	            //Waiting for new postion from input, then setting end position
	            IF #sx_TrigPECInfeedD
	                AND #iqUDT_RATPositioning.Upper.StartPositionD <> 0
	                AND ((#sx_DataReceived
	                AND NOT #sx_DestinationC)
	                OR NOT #sx_DataReceived)
	            THEN
	                #sx_ServoInfeed := TRUE;
	                #iqUDT_RATPositioning.Upper.EndPosition := #iqUDT_RATPositioning.Upper.StartPositionD - #iUDT_Configuration.InfeedDDistance;
	                #sx_TrigPECInfeedD := FALSE;
	                #iqUDT_RATPositioning.Upper.StartPositionD := 0;
	                #iqUDT_RATPositioning.Upper.PositionRequired := FALSE;
	                #iqUDT_RATPositioning.Upper.Start := TRUE;
	                // If straight destination detected then use displacement mode
	            ELSIF #sx_TrigPECInfeedD
	                AND #sx_DataReceived
	                AND #sx_DestinationC
	            THEN
	                #si_UpperInfeedDistance := ABS(#iUDT_Configuration.InfeedDDistance / 10);
	                #sx_TrigPECInfeedD := FALSE;
	                #sx_DisplacementInfeed := TRUE;
	                #iqUDT_RATPositioning.Upper.StartPositionD := 0;
	                #iqUDT_RATPositioning.Upper.PositionRequired := FALSE;
	            END_IF;

	            //If position is reached, set ProductRecived
	            IF #sR_TRIG_UpperInfeedDone.Q
	                AND #sx_ServoInfeed
	            THEN
	                #sx_ProductReceivedUp := TRUE;
	                #iqUDT_RATPositioning.Upper.Start := FALSE;
	            END_IF;

	            // During upper infeeding count distance to end of RAT
	            IF #sx_UpperTransportIn AND
	                #sx_DisplacementInfeed
	                AND NOT #sx_ProductReceivedUp
	            THEN
	                #si_UpperInfeedDistance -= ABS(#iqUDT_UpperConveyorInterface.Displacement);
	                IF #si_UpperInfeedDistance <= 0
	                THEN
	                    #sx_ProductReceivedUp := TRUE;
	                END_IF;
	            END_IF;

	        END_REGION

	    END_REGION

	    REGION 7.4 - Infeed checked, go to infeed level
	        // Lower
	        IF #sx_AutomaticActive                                          // The device is automaticly started
	            AND #sx_Ready                                               // The device is ready to opereate
	            AND #sx_Active                                              // The sequence is started
	            AND #sx_InfeedCHK                                           // Step infeed check is active
	            AND ((#si_Conveyor = #ci_ConveyorA) OR #si_Conveyor = #ci_ConveyorB)// Infeed is on low level
	        THEN
	            #sx_MoveSectionDownInfeed := TRUE;                          // Move section down
	            #sx_InfeedCHK := FALSE;                                     // Reset step infeed check
	            #si_Step := 2;                                              // Set step number for diagnostic purposes
	            // Upper
	        ELSIF #sx_AutomaticActive                                       // The device is automaticly started
	            AND #sx_Ready                                               // The device is ready to opereate
	            AND #sx_Active                                              // The sequence is started
	            AND #sx_InfeedCHK                                           // Step infeed check is active
	            AND ((#si_Conveyor = #ci_ConveyorC) OR #si_Conveyor = #ci_ConveyorD) // Infeed is on high level
	        THEN
	            #sx_MoveSectionUpinfeed := TRUE;                            // Move section up
	            #sx_InfeedCHK := FALSE;                                     // Reset step infeed check
	            #si_Step := 2;                                              // Set step number for diagnostic purposes
	        END_IF;
	    END_REGION

	    REGION 7.5 - At infeed level, start infeed transport
	        // Lower
	        IF #sx_AutomaticActive                                          // The device is automaticly started
	            AND #sx_Ready                                               // The device is ready to opereate
	            AND #sx_Active                                              // The sequence is started
	            AND (#ix_SectionIsDown                                      // Section is actual down
	            OR (#sx_SectionDown                                         // or request to go down is set and configuration allows it
	            AND NOT #iUDT_Configuration.PositionVerification))
	            AND #sx_MoveSectionDownInfeed                               // Step move down to infeed was activated
	        THEN
	            #sx_MoveSectionDownInfeed := FALSE;                         // Reset step move down to infeed level
	            #sx_LowerTransportIn := TRUE;                               // Start infeed roller transport
	            #iqUDT_RATPositioning.Lower.PositionRequired := TRUE;
	            #sx_LowerRTR := TRUE;                                       // Set RTR to infeed until TIP gets active
	            #si_Step := 3;                                              // Set step number for diagnostic purposes
	            // Upper
	        ELSIF #sx_AutomaticActive                                       // The device is automaticly started
	            AND #sx_Ready                                               // The device is ready to opereate
	            AND #sx_Active                                              // The sequence is started
	            AND (#ix_SectionIsUp                                        // Section is actual up
	            OR (#sx_SectionUp                                           // or request to go up is set and configuration allows it
	            AND NOT #iUDT_Configuration.PositionVerification))
	            AND #sx_MoveSectionUpinfeed                                 // Step move up to infeed was activated
	            //     AND #iqUDT_UpperConveyorInterface.ActualSpeed = 0
	        THEN
	            #sx_MoveSectionUpinfeed := FALSE;                           // Reset step move up to infeed level
	            #sx_UpperTransportIn := TRUE;                               // Start infeed belt transport
	            #iqUDT_RATPositioning.Upper.PositionRequired := TRUE;
	            #sx_UpperRTR := TRUE;                                       // Set RTR to infeed until TIP gets active
	            #si_Step := 3;                                              // Set step number for diagnostic purposes

	        END_IF;
	    END_REGION

	    REGION 7.6 - Stop transport, wait for destnation

	        // Lower
	        IF #sx_AutomaticActive                                          // The device is automaticly started
	            AND #sx_Ready                                               // The device is ready to opereate
	            AND #sx_Active                                              // The sequence is started
	            AND #sx_LowerTransportIn                                    // Step infeed lower transport is active
	            AND (NOT #sx_PECFiltered OR NOT #iUDT_Configuration.ControlProductWithPEC)                                     // Position is occupied
	            AND #sx_ProductReceivedDown                                // Product available at the end of RAT

	        THEN
	            #sx_LowerTransportIn := FALSE;                              // Reset step infeed lower transport
	            #sx_LowerRTR := FALSE;                                      // Reset RTR signal for infeed conveyor
	            #sx_UpDown := TRUE;                                         // Wait for direction
	            #sx_ProductReceivedDown := FALSE;                           // Reset "product received" bit
	            #sx_ServoInfeed := FALSE;
	            #sx_DisplacementInfeed := FALSE;
	            #si_Step := 4;                                              // Set step number for diagnostic purposes

	            // Upper
	        ELSIF #sx_AutomaticActive                                       // The device is automaticly started
	            AND #sx_Ready                                               // The device is ready to opereate
	            AND #sx_Active                                              // The sequence is started
	            AND #sx_UpperTransportIn                                    // Step infeed belt transport is active
	            AND (NOT #sx_PECFiltered OR NOT #iUDT_Configuration.ControlProductWithPEC)                                      // Position is occupied
	            AND #sx_ProductReceivedUp                                  // Product available at the end of RAT
	        THEN
	            #sx_UpperTransportIn := FALSE;                              // Reset step infeed belttransport
	            #sx_UpperRTR := FALSE;                                      // Reset RTR signal for infeed conveyor
	            #sx_UpDown := TRUE;                                         // Wait for direction
	            #sx_ProductReceivedUp := FALSE;                             // Reset "product received" bit
	            #sx_ServoInfeed := FALSE;
	            #sx_DisplacementInfeed := FALSE;
	            #si_Step := 4;                                              // Set step number for diagnostic purposes

	        END_IF;
	    END_REGION

	    REGION 7.7 - Destination received, move to outfeed level
	        IF #sx_AutomaticActive                                                  // The device is automaticly started
	            AND #sx_Ready                                                       // The device is ready to opereate
	            AND #sx_Active                                                      // The sequence is started
	            AND #sx_UpDown                                                      // Wait for direction
	            AND #sx_DataReceived                                                // Direction is received
	        THEN
	            #sx_UpDown := FALSE;                                                // Wait for direction
	            #sx_MoveSectionDownOutfeed := #sx_DestinationA OR #sx_DestinationB; // Depending on outfeed conveyor section is moved to outfeed level
	            #sx_MoveSectionUpOutfeed := #sx_DestinationC OR #sx_DestinationD;   // Depending on outfeed conveyor section is moved to outfeed level
	            #si_Step := 5;                                                      // Set step number for diagnostic purposes
	        END_IF;
	    END_REGION


	    REGION 7.8 - At outfeed level, start outfeed transport
	        // Lower
	        IF #sx_AutomaticActive                                          // The device is automaticly started
	            AND #sx_Ready                                               // The device is ready to opereate
	            AND #sx_Active                                              // The sequence is started
	            AND #sx_MoveSectionDownOutfeed                              // Step move down to outfeed is active
	            AND (#ix_SectionIsDown                                      // Section is actual down
	            OR (#sx_SectionDown                                         // or request to go down is set and configuration allows it
	            AND NOT #iUDT_Configuration.PositionVerification))
	        THEN
	            #sx_MoveSectionDownOutfeed := FALSE;                        // Reset step move down to outfeed
	            #sx_LowerTransportOut := TRUE;                              // Start outfeed roller transport
	            #si_LowerOutfeedDistance := DINT_TO_INT(#iUDT_LowerConveyorConfiguration.Common.Length / 10);
	            #si_Step := 6;                                              // Set step number for diagnostic purposes
	            // Upper
	        ELSIF #sx_AutomaticActive                                       // The device is automaticly started
	            AND #sx_Ready                                               // The device is ready to opereate
	            AND #sx_Active                                              // The sequence is startede
	            AND #sx_MoveSectionUpOutfeed                                // Step move up to outfeed is active
	            AND (#ix_SectionIsUp                                        // Section is actual up
	            OR (#sx_SectionUp                                          // or request to go up is set and configuration allows it
	            AND NOT #iUDT_Configuration.PositionVerification))
	        THEN
	            #sx_MoveSectionUpOutfeed := FALSE;                          // Reset step move up to outfeed
	            #sx_UpperTransportOut := TRUE;                              // Start outfeed belt transport
	            #si_UpperOutfeedDistance := DINT_TO_INT(#iUDT_UpperConveyorConfiguration.Common.Length / 10);
	            #si_Step := 6;                                              // Set step number for diagnostic purposes
	        END_IF;
	    END_REGION


	    REGION 7.9 Outfeed product tracking

	        IF #sx_LowerTransportOut AND NOT #sx_ProductSentDown
	        THEN
	            #si_LowerOutfeedDistance -= ABS(#iqUDT_LowerConveyorInterface.Displacement);
	            IF #si_LowerOutfeedDistance <= 0
	            THEN
	                #sx_ProductSentDown := TRUE;
	            END_IF;
	        END_IF;

	        // Upper
	        IF #sx_UpperTransportOut AND NOT #sx_ProductSentUp
	        THEN
	            #si_UpperOutfeedDistance -= ABS(#iqUDT_UpperConveyorInterface.Displacement);
	            IF #si_UpperOutfeedDistance <= 0
	            THEN
	                #sx_ProductSentUp := TRUE;
	            END_IF;
	        END_IF;

	    END_REGION

	    REGION 7.9 - End sequence
	        IF #sx_AutomaticActive                                          // The device is automaticly started
	            AND #sx_Ready                                               // The device is ready to opereate
	            AND #sx_Active                                              // The sequence is started
	            AND ((#sx_LowerTransportOut AND #sx_ProductSentDown)        // Outfeed transport is active and Produce is away
	            OR (#sx_UpperTransportOut AND #sx_ProductSentUp))           // Outfeed transport is active and Produce is away
	            AND (#sx_PECFiltered OR NOT #iUDT_Configuration.ControlProductWithPEC)                                          // Position is cleared
	            OR #sFB_InfeedTimeout.qx_DelayedSignal                      // Operation time elapsed
	        THEN

	            // Reset all auxiliary bits and variables
	            #sx_LowerTransportOut := FALSE;
	            #sx_UpperTransportOut := FALSE;
	            #si_Conveyor := 0;
	            #sx_Active := FALSE;
	            #sx_DataReceived := FALSE;
	            #si_Step := 0;
	            IF #sx_DestinationA
	            THEN
	                #sx_DestinationA := FALSE;
	                #iqUDT_HandShakeConveyorA.GIN := 0;
	                #iqUDT_HandShakeConveyorA.NrOfPosToShift := 0;
	                #iqUDT_HandShakeConveyorA.TIP := FALSE;
	            END_IF;
	            IF #sx_DestinationB
	            THEN
	                #sx_DestinationB := FALSE;
	                #iqUDT_HandShakeConveyorB.GIN := 0;
	                #iqUDT_HandShakeConveyorB.NrOfPosToShift := 0;
	                #iqUDT_HandShakeConveyorB.TIP := FALSE;
	            END_IF;
	            IF #sx_DestinationC
	            THEN
	                #sx_DestinationC := FALSE;
	                #iqUDT_HandShakeConveyorC.GIN := 0;
	                #iqUDT_HandShakeConveyorC.NrOfPosToShift := 0;
	                #iqUDT_HandShakeConveyorC.TIP := FALSE;
	            END_IF;
	            IF #sx_DestinationD
	            THEN
	                #sx_DestinationD := FALSE;
	                #iqUDT_HandShakeConveyorD.GIN := 0;
	                #iqUDT_HandShakeConveyorD.NrOfPosToShift := 0;
	                #iqUDT_HandShakeConveyorD.TIP := FALSE;
	            END_IF;
	            #iqUDT_HandShakeConveyorA.RTR := FALSE;
	            #iqUDT_HandShakeConveyorB.RTR := FALSE;
	            #iqUDT_HandShakeConveyorC.RTR := FALSE;
	            #iqUDT_HandShakeConveyorD.RTR := FALSE;

	            #si_Destination := 0;
	            #sx_ProductReceivedDown := FALSE;
	            #sx_ProductReceivedUp := FALSE;
	            #sx_ProductSentDown := FALSE;
	            #sx_ProductSentUp := FALSE;
	            #iqUDT_RATPositioning.Lower.ResetPosition := TRUE;
	            #iqUDT_RATPositioning.Upper.ResetPosition := TRUE;
	            #iqUDT_RATPositioning.Lower.StartPositionA := 0;
	            #iqUDT_RATPositioning.Lower.StartPositionB := 0;
	            #iqUDT_RATPositioning.Upper.StartPositionC := 0;
	            #iqUDT_RATPositioning.Upper.StartPositionD := 0;
	            #iqUDT_RATPositioning.Lower.PositionRequired := FALSE;
	            #iqUDT_RATPositioning.Upper.PositionRequired := FALSE;

	            // Move to configured default position
	            IF #iUDT_Configuration.DefaultPosition = #ci_DefaultPositionUp
	                AND #ix_SectionIsUp                                     // Section is actual up
	                AND #sa_FiFo[1] = 0
	            THEN
	                #sx_MoveSectiondownEnd := TRUE;                         // Then move down to infeed
	            END_IF;
	            IF #iUDT_Configuration.DefaultPosition = #ci_DefaultPositiondown
	                AND #ix_SectionIsDown                                   // Section is actual down
	                AND #sa_FiFo[1] = 0
	            THEN
	                #sx_MoveSectionUpEnd := TRUE;                           // Then move down to infeed
	            END_IF;
	        END_IF;
	        // Reset when on position
	        IF #sx_MoveSectionUpEnd                                         // Reset Up request when up
	            AND #ix_SectionIsUp
	        THEN
	            #sx_MoveSectionUpEnd := False;
	        END_IF;

	        IF #sx_MoveSectiondownEnd                                       // Reset down request when down
	            AND #ix_SectionIsDown
	        THEN
	            #sx_MoveSectiondownEnd := False;
	        END_IF;

	    END_REGION
	END_REGION

	REGION 8 - Output
	    REGION 8.1 - Lifting device

	        // Conditions to move sention down
	        #sx_SectionDown := (#sx_AutomaticActive
	        AND
	        ((#sx_MoveSectionDownInfeed OR #sx_MoveSectionDownOutfeed OR #sx_MoveSectiondownEnd))
	        OR (#sx_ManualModeActive AND #sx_ManualGoDown));
	        // Conditions to move sention up
	        #sx_SectionUp := (#sx_AutomaticActive
	        AND
	        ((#sx_MoveSectionUpinfeed OR #sx_MoveSectionUpOutfeed OR #sx_MoveSectionUpEnd))
	        OR (#sx_ManualModeActive AND #sx_ManualGoUp));

	        // Write valve outputs
	        IF #sx_SectionUp
	        THEN
	            #qx_PopupControl := TRUE;
	        ELSIF #sx_SectionDown
	        THEN
	            #qx_PopupControl := FALSE;
	        END_IF;

	    END_REGION

	    REGION 8.2 - Lower conveyor

	        // Run forward
	        #tx_LowerConveyorRunFwd :=
	        ((#sx_LowerTransportIn AND (#si_Conveyor = #ci_ConveyorA) AND #ix_ConveyorAAuto)                                    // Transport in and transporting from infeed A
	        OR (#sx_LowerTransportOut AND #sx_DestinationB AND #iqUDT_HandShakeConveyorB.RTR))                      // Transport out and RTR is received
	        AND #sx_AutomaticActive;

	        // Run reverse
	        #tx_LowerConveyorRunRvs :=
	        ((#sx_LowerTransportIn AND (#si_Conveyor = #ci_ConveyorB) AND #ix_ConveyorBAuto)                                     // Transport in and transporting from infeed B
	        OR (#sx_LowerTransportOut AND #sx_DestinationA AND #iqUDT_HandShakeConveyorA.RTR))                      // Transport out AND RTR is received
	        AND #sx_AutomaticActive;
	        // Handshake RTR mapping
	        #sUDT_HandshakeUpLowerConveyor.RTR := #tx_LowerConveyorRunRvs;
	        #sUDT_HandshakeLowerConveyor.RTR := #tx_LowerConveyorRunFwd;

	        IF #tx_LowerConveyorRunRvs THEN
	            #sx_ReverseLower := TRUE;
	        END_IF;

	        IF #tx_LowerConveyorRunFwd THEN
	            #sx_ReverseLower := FALSE;
	        END_IF;

	        // Control lower conveyor with FB_Conveyor block
	        #sFB_Conveyor_LowerConveyor(iUDT_ConveyorConfiguration := #iUDT_LowerConveyorConfiguration,
	                                    ix_SafetyOk := #ix_SafetyOk,
	                                    ix_24vOk := #ix_24vOk,
	                                    ix_400vOk := #ix_400vOk,
	                                    ix_HardwareOk := #ix_HardwareOk,
	                                    ix_ReverseDirection := #sx_ReverseLower,
	                                    ix_ResetEnergySave := TRUE,
	                                    qUDT_HMIStatus => #qUDT_HMIConveyorStatus,
	                                    qUDT_Status => #qUDT_ConveyorStatus,
	                                    iqUDT_EquipmentControl := #iqUDT_EquipmentControl,
	                                    iqUDT_ConveyorCommand := #iqUDT_ConveyorCommand,
	                                    iqUDT_ConveyorInterface := #iqUDT_LowerConveyorInterface,
	                                    iqUDT_HandShakeUp := #sUDT_HandshakeUpLowerConveyor,
	                                    iqUDT_HandShake := #sUDT_HandshakeLowerConveyor,
	                                    iqUDT_Statistics := #iqUDT_ConveyorStatistics);

	    END_REGION

	    REGION 8.3 - Upper conveyor

	        // Run forward
	        #tx_UpperConveyorRunFwd :=
	        ((#sx_UpperTransportIn AND (#si_Conveyor = #ci_ConveyorC) AND #ix_ConveyorCAuto)                                                  // Transport in and transporting from infeed C c
	        OR (#sx_UpperTransportOut AND #sx_DestinationD AND #iqUDT_HandShakeConveyorD.RTR))             // Transport out and RTR is received
	        AND #sx_AutomaticActive;

	        // Run reverse
	        #tx_UpperConveyorRunRvs :=
	        ((#sx_UpperTransportIn AND (#si_Conveyor = #ci_ConveyorD) AND #ix_ConveyorDAuto)                                                   // Transport in and transporting from infeed D
	        OR (#sx_UpperTransportOut AND #sx_DestinationC AND #iqUDT_HandShakeConveyorC.RTR))              // Transport out and RTR is received
	        AND #sx_AutomaticActive;

	        // Handshake RTR mapping
	        #sUDT_HandshakeUpUpperConveyor.RTR := #tx_UpperConveyorRunRvs;
	        #sUDT_HandshakeUpperConveyor.RTR := #tx_UpperConveyorRunFwd;


	        // MAnual mode mapping from RAT structure
	        #tUDT_ConveyorCommandUpper.ManualMode := #iqUDT_RATCommand.ManualMode;
	        #tUDT_ConveyorCommandUpper.ManualStartStop := #iqUDT_RATCommand.ManualStartStop;
	        #tUDT_ConveyorCommandUpper.ManualFullSpeed := #iqUDT_RATCommand.ManualFullSpeed;
	        #tUDT_ConveyorCommandUpper.ManualSpeed := #iqUDT_RATCommand.ManualSpeed;
	        #tUDT_ConveyorCommandUpper.ManualJog := #iqUDT_RATCommand.ManualJog;
	        #tUDT_ConveyorCommandUpper.Reverse := #iqUDT_RATCommand.Reverse;

	        IF #tx_UpperConveyorRunRvs
	        THEN
	            #sx_ReverseUpper := TRUE;
	        END_IF;

	        IF #tx_UpperConveyorRunFwd
	        THEN
	            #sx_ReverseUpper := FALSE;
	        END_IF;

	        // Control pop-up conveyor with FB_Conveyor block
	        #sFB_Conveyor_UpperConveyor(iUDT_ConveyorConfiguration := #iUDT_UpperConveyorConfiguration,
	                                    ix_SafetyOk := #ix_SafetyOk,
	                                    ix_24vOk := #ix_24vOk,
	                                    ix_400vOk := #ix_400vOk,
	                                    ix_HardwareOk := #ix_HardwareOk,
	                                    ix_ReverseDirection := #sx_ReverseUpper,
	                                    ix_ExternalRequestDieBack := FALSE,
	                                    ix_ResetEnergySave := TRUE,
	                                    qUDT_HMIStatus => #tUDT_HMIStatus,
	                                    qUDT_Status => #tUDT_CommonStatus,
	                                    iqUDT_EquipmentControl := #iqUDT_EquipmentControl,
	                                    iqUDT_ConveyorCommand := #tUDT_ConveyorCommandUpper,
	                                    iqUDT_ConveyorInterface := #iqUDT_UpperConveyorInterface,
	                                    iqUDT_HandShakeUp := #sUDT_HandshakeUpUpperConveyor,
	                                    iqUDT_HandShake := #sUDT_HandshakeUpperConveyor,
	                                    iqUDT_Statistics := #tUDT_ConveyorStatistics);

	        // Manual mode mapping from conveyor to RAT
	        #iqUDT_RATCommand.ManualMode := #tUDT_ConveyorCommandUpper.ManualMode;
	        #iqUDT_RATCommand.ManualStartStop := #tUDT_ConveyorCommandUpper.ManualStartStop;
	        #iqUDT_RATCommand.ManualFullSpeed := #tUDT_ConveyorCommandUpper.ManualFullSpeed;
	        #iqUDT_RATCommand.ManualSpeed := #tUDT_ConveyorCommandUpper.ManualSpeed;
	        #iqUDT_RATCommand.ManualJog := #tUDT_ConveyorCommandUpper.ManualJog;

	    END_REGION


	    REGION 8.4 - Handshake in-outfeed conveyors

	        #iqUDT_HandShakeConveyorA.RTR := FALSE;
	        #iqUDT_HandShakeConveyorB.RTR := FALSE;
	        #iqUDT_HandShakeConveyorC.RTR := FALSE;
	        #iqUDT_HandShakeConveyorD.RTR := FALSE;

	        IF (#si_Conveyor = 1)
	        THEN
	            // Infeed conveyor low level
	            #iqUDT_HandShakeConveyorA.CascadeStartUp := #sx_AutomaticActive;
	            #iqUDT_HandShakeConveyorA.RTR := (#sx_LowerRTR OR #iqUDT_HandShakeConveyorA.TIP) AND #sx_AutomaticActive;
	            #iqUDT_HandShakeConveyorA.ResetEnergySave := false;

	            IF #sx_LowerTransportIn
	            THEN
	                IF #iqUDT_HandShakeConveyorA.GIN <> 0
	                THEN                          // Save gin number in buffer
	                    #sUDT_HandshakeBuffer.GIN := #iqUDT_HandShakeConveyorA.GIN;
	                END_IF;

	                // Count number position to shift in buffer
	                #sUDT_HandshakeBuffer.NrOfPosToShift += #iqUDT_HandShakeConveyorA.NrOfPosToShift;
	                #iqUDT_HandShakeConveyorA.NrOfPosToShift := 0;
	            END_IF;

	        ELSE
	            // Outfeed conveyor low level
	            #qx_ExternalSendRequestA := #sx_DestinationA AND NOT #sFB_PEC.qx_PECFiltered;// AND #sx_LowerTransportOut;
	            IF #sx_LowerTransportOut AND #sx_DestinationA
	            THEN
	                IF #sR_TRIG_LowerOutfeedRunning.Q
	                THEN
	                    #iqUDT_HandShakeConveyorA.GIN := #sUDT_HandshakeBuffer.GIN;
	                    #iqUDT_HandShakeConveyorA.NrOfPosToShift := #sUDT_HandshakeBuffer.NrOfPosToShift;
	                    #sUDT_HandshakeBuffer.GIN := 0;
	                    #sUDT_HandshakeBuffer.NrOfPosToShift := 0;
	                END_IF;

	                IF #ix_PEC
	                THEN
	                    #iqUDT_HandShakeConveyorA.GIN := 0;
	                    #iqUDT_HandShakeConveyorA.NrOfPosToShift := 0;
	                END_IF;
	            END_IF;

	        END_IF;

	        IF (#si_Conveyor = 2)
	        THEN
	            // Infeed conveyor low level
	            #iqUDT_HandShakeConveyorB.CascadeStartUp := #sx_AutomaticActive;
	            #iqUDT_HandShakeConveyorB.RTR := (#sx_LowerRTR OR #iqUDT_HandShakeConveyorB.TIP) AND #sx_AutomaticActive;
	            #iqUDT_HandShakeConveyorB.ResetEnergySave := false;
	            IF #sx_LowerTransportIn
	            THEN
	                IF #iqUDT_HandShakeConveyorB.GIN <> 0
	                THEN
	                    #sUDT_HandshakeBuffer.GIN := #iqUDT_HandShakeConveyorB.GIN;
	                END_IF;

	                #sUDT_HandshakeBuffer.NrOfPosToShift += #iqUDT_HandShakeConveyorB.NrOfPosToShift;
	                #iqUDT_HandShakeConveyorB.NrOfPosToShift := 0;
	            END_IF;
	        ELSE
	            // Outfeed conveyor low level
	            #qx_ExternalSendRequestB := #sx_DestinationB AND NOT #sFB_PEC.qx_PECFiltered;// AND #sx_LowerTransportOut;
	            IF #sx_DestinationB AND #sx_LowerTransportOut
	            THEN
	                IF #sR_TRIG_LowerOutfeedRunning.Q
	                THEN
	                    #iqUDT_HandShakeConveyorB.GIN := #sUDT_HandshakeBuffer.GIN;
	                    #iqUDT_HandShakeConveyorB.NrOfPosToShift := #sUDT_HandshakeBuffer.NrOfPosToShift;
	                    #sUDT_HandshakeBuffer.GIN := 0;
	                    #sUDT_HandshakeBuffer.NrOfPosToShift := 0;
	                END_IF;

	                IF #ix_PEC
	                THEN
	                    #iqUDT_HandShakeConveyorB.GIN := 0;
	                    #iqUDT_HandShakeConveyorB.NrOfPosToShift := 0;

	                END_IF;

	            END_IF;
	        END_IF;

	        IF (#si_Conveyor = 3)
	        THEN
	            // Infeed conveyor high level
	            #iqUDT_HandShakeConveyorC.CascadeStartUp := #sx_AutomaticActive;
	            #iqUDT_HandShakeConveyorC.RTR := (#sx_UpperRTR OR #iqUDT_HandShakeConveyorC.TIP) AND #sx_AutomaticActive;
	            #iqUDT_HandShakeConveyorC.ResetEnergySave := false;
	            IF #sx_UpperTransportIn
	            THEN
	                IF #iqUDT_HandShakeConveyorC.GIN <> 0
	                THEN
	                    #sUDT_HandshakeBuffer.GIN := #iqUDT_HandShakeConveyorC.GIN;
	                END_IF;

	                #sUDT_HandshakeBuffer.NrOfPosToShift += #iqUDT_HandShakeConveyorC.NrOfPosToShift;
	                #iqUDT_HandShakeConveyorC.NrOfPosToShift := 0;
	            END_IF;
	        ELSE
	            // Outfeed conveyor high level
	            #qx_ExternalSendRequestC := #sx_DestinationC AND NOT #sFB_PEC.qx_PECFiltered;// AND #sx_LowerTransportOut;
	            IF #sx_DestinationC AND #sx_UpperTransportOut
	            THEN
	                IF #sR_TRIG_UpperOutfeedRunning.Q
	                THEN
	                    #iqUDT_HandShakeConveyorC.GIN := #sUDT_HandshakeBuffer.GIN;
	                    #iqUDT_HandShakeConveyorC.NrOfPosToShift := #sUDT_HandshakeBuffer.NrOfPosToShift;
	                    #sUDT_HandshakeBuffer.GIN := 0;
	                    #sUDT_HandshakeBuffer.NrOfPosToShift := 0;
	                END_IF;
	                IF #ix_PEC
	                THEN
	                    #iqUDT_HandShakeConveyorC.GIN := 0;
	                    #iqUDT_HandShakeConveyorC.NrOfPosToShift := 0;
	                END_IF;

	            END_IF;

	        END_IF;

	        IF (#si_Conveyor = 4)
	        THEN
	            // Infeed conveyor high level
	            #iqUDT_HandShakeConveyorD.CascadeStartUp := #sx_AutomaticActive;
	            #iqUDT_HandShakeConveyorD.RTR := (#sx_UpperRTR OR #iqUDT_HandShakeConveyorD.TIP) AND #sx_AutomaticActive;
	            #iqUDT_HandShakeConveyorD.ResetEnergySave := false;
	            IF #sx_UpperTransportIn
	            THEN
	                IF #iqUDT_HandShakeConveyorD.GIN <> 0
	                THEN
	                    #sUDT_HandshakeBuffer.GIN := #iqUDT_HandShakeConveyorD.GIN;
	                END_IF;

	                #sUDT_HandshakeBuffer.NrOfPosToShift += #iqUDT_HandShakeConveyorD.NrOfPosToShift;
	                #iqUDT_HandShakeConveyorD.NrOfPosToShift := 0;
	            END_IF;
	        ELSE
	            // Outfeed conveyor high level
	            #qx_ExternalSendRequestD := #sx_DestinationD AND NOT #sFB_PEC.qx_PECFiltered;// AND #sx_LowerTransportOut;
	            IF #sx_DestinationD AND #sx_UpperTransportOut
	            THEN
	                IF #sR_TRIG_UpperOutfeedRunning.Q
	                THEN
	                    #iqUDT_HandShakeConveyorD.GIN := #sUDT_HandshakeBuffer.GIN;
	                    #iqUDT_HandShakeConveyorD.NrOfPosToShift := #sUDT_HandshakeBuffer.NrOfPosToShift;
	                    #sUDT_HandshakeBuffer.GIN := 0;
	                    #sUDT_HandshakeBuffer.NrOfPosToShift := 0;
	                END_IF;

	                IF #ix_PEC
	                THEN
	                    #iqUDT_HandShakeConveyorD.GIN := 0;
	                    #iqUDT_HandShakeConveyorD.NrOfPosToShift := 0;
	                END_IF;

	            END_IF;

	        END_IF;

	    END_REGION

	    REGION 8.5 - Blade stop EoS
	        // If blade stop is available then handle valve
	        IF #iUDT_Configuration.BladeStopEoS
	        THEN
	            // Use blade stop if product is comming from A to side destination
	            IF #si_Conveyor = #ci_ConveyorA AND (#sx_DestinationC OR #sx_DestinationD) AND #sx_LowerTransportIn
	            THEN
	                #sx_BladeStopEoSControl := TRUE;
	            END_IF;
	            IF NOT #sx_LowerTransportIn
	            THEN
	                #sx_BladeStopEoSControl := FALSE;
	            END_IF;
	            #iqUDT_BladeStopEoSInterface.Open := #sx_BladeStopEoSControl;
	        END_IF;

	    END_REGION

	    REGION 8.6 - Blade stop BoS
	        IF #iUDT_Configuration.BladeStopBoS
	        THEN
	            // Use blade stop if product is comming from B to side destination
	            IF #si_Conveyor = #ci_ConveyorB AND (#sx_DestinationC OR #sx_DestinationD) AND #sx_LowerTransportIn
	            THEN
	                #sx_BladeStopBoSControl := TRUE;
	            END_IF;
	            IF NOT #sx_LowerTransportIn
	            THEN
	                #sx_BladeStopBoSControl := FALSE;
	            END_IF;
	            #iqUDT_BladeStopBoSInterface.Open := #sx_BladeStopBoSControl;
	        END_IF;

	    END_REGION

	END_REGION

	REGION 9 - PEC
	    // Use displacement from both interfaces - lower and upper
	    #tUDT_ConveyorInterface := #iqUDT_UpperConveyorInterface;
	    #tUDT_ConveyorInterface.Displacement := #iqUDT_UpperConveyorInterface.Displacement + #iqUDT_LowerConveyorInterface.Displacement;

	    // PEC handling
	    #sFB_PEC(ix_PEC := #ix_PEC,
	             iUDT_PECConfiguration := #iUDT_PECConfiguration,
	             qUDT_HMIStatus => #qUDT_HMIPECStatus,
	             iqUDT_ConveyorInterface := #tUDT_ConveyorInterface,
	             iqUDT_PECStatistics := #iqUDT_PECStatistics);

	    // copy error to both intefaces - lower and upper
	    #iqUDT_UpperConveyorInterface.InternalErrorPEC := #iqUDT_UpperConveyorInterface.InternalErrorPEC OR #tUDT_ConveyorInterface.InternalErrorPEC;
	    #iqUDT_LowerConveyorInterface.InternalErrorPEC := #iqUDT_LowerConveyorInterface.InternalErrorPEC OR #tUDT_ConveyorInterface.InternalErrorPEC;

	END_REGION

	REGION 9 - Status

	    // Status update
	    #sUDT_HMIStatus.Specific.Down := #ix_SectionIsDown AND NOT #ix_SectionIsUp;
	    #sUDT_HMIStatus.Specific.Up := #ix_SectionIsUp AND NOT #ix_SectionIsDown;
	    #sUDT_HMIStatus.Specific.Reverse := #tUDT_HMIStatus.Specific.Reverse;
	    #sUDT_HMIStatus.Status := #tUDT_HMIStatus.Status;

	    #sUDT_CommonStatus.SafetyStop := NOT #ix_SafetyOk AND #ix_HardwareOk;
	    #sUDT_CommonStatus.Stopped := NOT #sx_Ready OR NOT #sx_AutomaticActive OR #tUDT_CommonStatus.Stopped;
	    #sUDT_CommonStatus.AutoON := #sx_Ready AND #sx_AutomaticActive AND #tUDT_CommonStatus.AutoON;
	    #sUDT_CommonStatus.Manual := #sx_ManualModeActive;
	    #sUDT_CommonStatus.ManualRun := #sx_ManualModeActive AND #sUDT_CommonStatus.Running;
	    #sUDT_CommonStatus.Running := #tUDT_CommonStatus.Running;

	    #qUDT_RATStatus := #sUDT_CommonStatus;
	    #qUDT_HMIRATStatus := #sUDT_HMIStatus;

	END_REGION

	REGION 10 - Statistics

	    REGION 10.1 - Air pressure fault
	        // Update statistics if error is active or statistics reset detected
	        IF #sUDT_HMIStatus.Specific.ErrAirpressureNotOk OR #iqUDT_EquipmentControl.Command.ResetData      // Reset statistics
	        THEN

	            "FC_Statistics"(ix_Reset := #iqUDT_EquipmentControl.Command.ResetData,  // Reset statistics input
	                            ix_Activate := #sUDT_HMIStatus.Specific.ErrAirpressureNotOk,
	                            ix_RTrigActivate := #sR_TRIG_AirPressureFault.Q,            // Statistics active trigger
	                            iqUDT_Statistics := #iqUDT_RATStatistics.AirPressure);

	        END_IF;

	    END_REGION

	    REGION 10.2 - Device up time

	        // Conveyor up is when conveyor is not in manual mode and has an error
	        IF #sx_DivertUpRunTimeErr OR #iqUDT_EquipmentControl.Command.ResetData      // Reset statistics
	        THEN

	            "FC_Statistics"(ix_Reset := #iqUDT_EquipmentControl.Command.ResetData,  // Reset statistics input
	                            ix_Activate := #sx_DivertUpRunTimeErr, // Activate statistics functions input
	                            ix_RTrigActivate := #sR_TRIG_DivertUpError.Q,          // Statistics active trigger
	                            iqUDT_Statistics := #iqUDT_RATStatistics.DivertUpError);   // Statistics values output

	        END_IF;

	    END_REGION

	    REGION 10.3 - Device down time

	        // Conveyor down is when conveyor is not in manual mode and has an error
	        IF #sx_DivertDownRunTimeErr OR #iqUDT_EquipmentControl.Command.ResetData      // Reset statistics
	        THEN

	            "FC_Statistics"(ix_Reset := #iqUDT_EquipmentControl.Command.ResetData,  // Reset statistics input
	                            ix_Activate := #sx_DivertDownRunTimeErr, // Activate statistics functions input
	                            ix_RTrigActivate := #sR_TRIG_DivertDownError.Q,          // Statistics active trigger
	                            iqUDT_Statistics := #iqUDT_RATStatistics.DivertDownError);   // Statistics values output

	        END_IF;

	    END_REGION

	    REGION 10.4 - Conveyor statistics
	        // Copy statistics from conveyor block
	        #iqUDT_RATStatistics.ConveyorDown := #tUDT_ConveyorStatistics.ConveyorDown;
	        #iqUDT_RATStatistics.ConveyorStop := #tUDT_ConveyorStatistics.ConveyorStop;
	        #iqUDT_RATStatistics.ConveyorUp := #tUDT_ConveyorStatistics.ConveyorUp;

	    END_REGION

	END_REGION

	REGION 11 - Report to control block
	    // Function to manage report between control block and conveyor block
	    "FC_EquipmentReport"(iUDT_Status := #sUDT_CommonStatus,
	                         iqUDT_Control := #iqUDT_EquipmentControl);

	END_REGION

	REGION 12 - Internal errors and warnings reset

	    REGION 12.1 Infeed timeout
	        // Infeed stuck, timeout calculation
	        #sFB_InfeedTimeout(iudi_OnDelayTime := #iUDT_Configuration.InfeedTimeout,
	                           ix_SignalToDelay := #si_Step = 3 AND (#sx_ProductReceivedDown OR #sx_ProductReceivedUp));

	    END_REGION

	    REGION 12.2 Reactivation
	        // Reactivate conveyor 1 if request is active and no register find
	        #sFB_ConveyorAReactivation(iudi_OnDelayTime := #iUDT_Configuration.ReactivationTime,
	                                   ix_SignalToDelay := #ix_ExternalReceiveRequestA AND #ix_ConveyorAAuto);

	        IF #sFB_ConveyorAReactivation.qx_DelayedSignal AND NOT (#si_Conveyor = 1)
	        THEN
	            #sx_ReactivateA := TRUE;
	            FOR #si_LoopArrayCount := 1 TO #ci_FiFoLength DO

	                IF #sa_FiFo[#si_LoopArrayCount] = 1
	                THEN
	                    #sx_ReactivateA := FALSE;
	                END_IF;

	            END_FOR;

	        END_IF;
	        // Reactivate conveyor 1 if request is active and no register find
	        #sFB_ConveyorBReactivation(iudi_OnDelayTime := #iUDT_Configuration.ReactivationTime,
	                                   ix_SignalToDelay := #ix_ExternalReceiveRequestB AND #ix_ConveyorBAuto);

	        IF #sFB_ConveyorBReactivation.qx_DelayedSignal AND NOT (#si_Conveyor = 2)
	        THEN
	            #sx_ReactivateB := TRUE;
	            FOR #si_LoopArrayCount := 1 TO #ci_FiFoLength DO

	                IF #sa_FiFo[#si_LoopArrayCount] = 2
	                THEN
	                    #sx_ReactivateB := FALSE;
	                END_IF;

	            END_FOR;

	        END_IF;
	        // Reactivate conveyor 1 if request is active and no register find
	        #sFB_ConveyorCReactivation(iudi_OnDelayTime := #iUDT_Configuration.ReactivationTime,
	                                   ix_SignalToDelay := #ix_ExternalReceiveRequestC AND #ix_ConveyorCAuto);

	        IF #sFB_ConveyorCReactivation.qx_DelayedSignal AND NOT (#si_Conveyor = 3)
	        THEN
	            #sx_ReactivateC := TRUE;
	            FOR #si_LoopArrayCount := 1 TO #ci_FiFoLength DO

	                IF #sa_FiFo[#si_LoopArrayCount] = 3
	                THEN
	                    #sx_ReactivateC := FALSE;
	                END_IF;

	            END_FOR;

	        END_IF;
	        // Reactivate conveyor 1 if request is active and no register find
	        #sFB_ConveyorDReactivation(iudi_OnDelayTime := #iUDT_Configuration.ReactivationTime,
	                                   ix_SignalToDelay := #ix_ExternalReceiveRequestD AND #ix_ConveyorDAuto);

	        IF #sFB_ConveyorDReactivation.qx_DelayedSignal AND NOT (#si_Conveyor = 4)
	        THEN
	            #sx_ReactivateD := TRUE;
	            FOR #si_LoopArrayCount := 1 TO #ci_FiFoLength DO

	                IF #sa_FiFo[#si_LoopArrayCount] = 4
	                THEN
	                    #sx_ReactivateD := FALSE;
	                END_IF;

	            END_FOR;

	        END_IF;

	    END_REGION

	END_REGION
END_FUNCTION_BLOCK

DATA_BLOCK "DB_FIFOLostGIN"
TITLE = DB_FIFO
{ S7_Optimized_Access := 'TRUE' }
AUTHOR : MHSE
FAMILY : GeneralSystemFunctions
VERSION : 3.0
NON_RETAIN
//Data block to store FIFO registers.
   VAR RETAIN
      Header { ExternalAccessible := 'False'; ExternalVisible := 'False'; ExternalWritable := 'False'; S7_SetPoint := 'False'} : "UDT_FifoHeader";   // FIFO Header
      Data { ExternalAccessible := 'False'; ExternalVisible := 'False'; ExternalWritable := 'False'} : Array[0..199] of Int;   // FIFO data buffer
   END_VAR
   VAR
      Header_1 { ExternalAccessible := 'False'; ExternalVisible := 'False'; ExternalWritable := 'False'; S7_SetPoint := 'False'} : "UDT_FifoHeader";
      Data_1 { ExternalAccessible := 'False'; ExternalVisible := 'False'; ExternalWritable := 'False'} : Array[0..199] of Int;
      Header_2 { ExternalAccessible := 'False'; ExternalVisible := 'False'; ExternalWritable := 'False'; S7_SetPoint := 'False'} : "UDT_FifoHeader";
      Data_2 { ExternalAccessible := 'False'; ExternalVisible := 'False'; ExternalWritable := 'False'} : Array[0..199] of Int;
      Header_3 { ExternalAccessible := 'False'; ExternalVisible := 'False'; ExternalWritable := 'False'; S7_SetPoint := 'False'} : "UDT_FifoHeader";
      Data_3 { ExternalAccessible := 'False'; ExternalVisible := 'False'; ExternalWritable := 'False'} : Array[0..199] of Int;
      Header_4 { ExternalAccessible := 'False'; ExternalVisible := 'False'; ExternalWritable := 'False'; S7_SetPoint := 'False'} : "UDT_FifoHeader";
      Data_4 { ExternalAccessible := 'False'; ExternalVisible := 'False'; ExternalWritable := 'False'} : Array[0..199] of Int;
      Header_5 { ExternalAccessible := 'False'; ExternalVisible := 'False'; ExternalWritable := 'False'; S7_SetPoint := 'False'} : "UDT_FifoHeader";
      Data_5 { ExternalAccessible := 'False'; ExternalVisible := 'False'; ExternalWritable := 'False'} : Array[0..199] of Int;
      Header_6 { ExternalAccessible := 'False'; ExternalVisible := 'False'; ExternalWritable := 'False'; S7_SetPoint := 'False'} : "UDT_FifoHeader";
      Data_6 { ExternalAccessible := 'False'; ExternalVisible := 'False'; ExternalWritable := 'False'} : Array[0..199] of Int;
   END_VAR


BEGIN

END_DATA_BLOCK

FUNCTION_BLOCK "FB_CognexDM260"
{ S7_Optimized_Access := 'TRUE' }
VERSION : 0.1
// ATTRIBUTES
// AUTO_NUMBER = True
// BLOCK_NUMBER = 263
// END_ATTRIBUTES
   VAR_INPUT
      iUDT_CognexDM260_IN { ExternalAccessible := 'False'; ExternalVisible := 'False'; ExternalWritable := 'False'} : "UDT_CognexDM260_IN";   // Data from camera
      ix_Trigger { ExternalAccessible := 'False'; ExternalVisible := 'False'; ExternalWritable := 'False'} : Bool;   // Trigger - Activate barcode scanning inside this function
   END_VAR

   VAR_OUTPUT
      qUDT_CognexDM260_OUT { ExternalAccessible := 'False'; ExternalVisible := 'False'; ExternalWritable := 'False'} : "UDT_CognexDM260_OUT";   // Data send to camera
      qs_Barcode { ExternalAccessible := 'False'; ExternalVisible := 'False'; ExternalWritable := 'False'} : String;
      qw_RetVal { ExternalAccessible := 'False'; ExternalVisible := 'False'; ExternalWritable := 'False'} : Word;   // Error code (W#16#...): A - TimeOut; B - Bit from camera "Result available" blocked; C - NO READ; C5 - 5 NO READ in row;  C0 - Empty data from camera
   END_VAR

   VAR_IN_OUT
      iqUDT_EquipmentControl { S7_HiddenAssignment := 'HideIfNoParamAssigned'} : "UDT_EquipmentControl";   // Optional. Use UDT to reset errors and statistic [ or two next bits:  ix_ResetError  to reset erors and ResetStatistic]
   END_VAR

   VAR
      sFB_TimerOnOffDelay_TimeOut { ExternalAccessible := 'False'; ExternalVisible := 'False'; ExternalWritable := 'False'; S7_SetPoint := 'False'} : "FB_TimerOnOffDelay";   // TimeOut timer
      sFB_TimerOnOffDelay_ResultsAvailableError { ExternalAccessible := 'False'; ExternalVisible := 'False'; ExternalWritable := 'False'; S7_SetPoint := 'False'} : "FB_TimerOnOffDelay";   // Timer for control Result Avilable duration time
      sFB_TimerOnOffDelay_ActTimeToNextReady { ExternalAccessible := 'False'; ExternalVisible := 'False'; ExternalWritable := 'False'; S7_SetPoint := 'False'} : "FB_TimerOnOffDelay";   // Time from trigger to get data from camera (Result_Available)
      sFB_TimerOnOffDelay_ActReadingFromCameraTime { ExternalAccessible := 'False'; ExternalVisible := 'False'; ExternalWritable := 'False'; S7_SetPoint := 'False'} : "FB_TimerOnOffDelay";   // Time from trigger to get data from camera (Result_Available)
      sR_TRIG_StatisticActCycleTime {InstructionName := 'R_TRIG'; LibVersion := '1.0'; ExternalAccessible := 'False'; ExternalVisible := 'False'; ExternalWritable := 'False'; S7_SetPoint := 'False'} : R_TRIG;   // Rising edge for (#R_TRIG_Result_available.Q OR #sx_ErrorTimeOut)
      sR_TRIG_Trigger {InstructionName := 'R_TRIG'; LibVersion := '1.0'; ExternalAccessible := 'False'; ExternalVisible := 'False'; ExternalWritable := 'False'; S7_SetPoint := 'False'} : R_TRIG;   // Rising edge trigger signal
      sR_TRIG_TriggerReady {InstructionName := 'R_TRIG'; LibVersion := '1.0'; ExternalAccessible := 'False'; ExternalVisible := 'False'; ExternalWritable := 'False'; S7_SetPoint := 'False'} : R_TRIG;   // Rising edge for bit from camera "trigger ready"
      sR_TRIG_ResultAvailable {InstructionName := 'R_TRIG'; LibVersion := '1.0'; ExternalAccessible := 'False'; ExternalVisible := 'False'; ExternalWritable := 'False'; S7_SetPoint := 'False'} : R_TRIG;   // Rising edge for bit from camera "Result_Available"
      sR_TRIG_NoReadCounter {InstructionName := 'R_TRIG'; LibVersion := '1.0'; ExternalAccessible := 'False'; ExternalVisible := 'False'; ExternalWritable := 'False'; S7_SetPoint := 'False'} : R_TRIG;   // Rising edge for general counter NO_READ
      sR_TRIG_OkReadCounter {InstructionName := 'R_TRIG'; LibVersion := '1.0'; ExternalAccessible := 'False'; ExternalVisible := 'False'; ExternalWritable := 'False'; S7_SetPoint := 'False'} : R_TRIG;   // Rising edge for general counter OK_READ
      sR_TRIG_TimeOutCounter {InstructionName := 'R_TRIG'; LibVersion := '1.0'; ExternalAccessible := 'False'; ExternalVisible := 'False'; ExternalWritable := 'False'; S7_SetPoint := 'False'} : R_TRIG;   // Rising edge for general counter TimeOut
      sR_TRIG_ResetStatistics {InstructionName := 'R_TRIG'; LibVersion := '1.0'; ExternalAccessible := 'False'; ExternalVisible := 'False'; ExternalWritable := 'False'; S7_SetPoint := 'False'} : R_TRIG;   // Rising edge for ResetStatistics
      ss_LastResults { ExternalAccessible := 'False'; ExternalVisible := 'False'; ExternalWritable := 'False'} : Struct   // Copy of last result reading barcode value
         ID { ExternalAccessible := 'False'; ExternalVisible := 'False'; ExternalWritable := 'False'} : Int;   // The value of the “Trigger ID” when the trigger that generated these results was issued. Used to match up triggers with corresponding result data (16-bit Integer).
         Flags { ExternalAccessible := 'False'; ExternalVisible := 'False'; ExternalWritable := 'False'} : Int;   // Indicates the success or failure of the read that produced these results (16-bit Integer).Bit 0,1=read, 0=no read, Bit 1,1=validated, 0=not validated (or validation not in use),  Bit 2,1=verified, 0=not verified (or verification not in use)  Bit 3,1=acquisition trigger overrun  Bit 4,1=acquisition buffer overflow
         Length { ExternalAccessible := 'False'; ExternalVisible := 'False'; ExternalWritable := 'False'} : Int;   // Actual number of bytes of read data contained in the “Result Data” field (16-bitInteger).
         DataBarCode { ExternalAccessible := 'False'; ExternalVisible := 'False'; ExternalWritable := 'False'} : Array[0..63] of Char;   // Last barcode
         DataBarCodeString { ExternalAccessible := 'False'; ExternalVisible := 'False'; ExternalWritable := 'False'} : String;   // Last barcode as string // for future use
      END_STRUCT;
      ss_Statistic { ExternalAccessible := 'False'; ExternalVisible := 'False'; ExternalWritable := 'False'} : Struct   // All statistics
         udi_ActReadingFromCameraTime { ExternalAccessible := 'False'; ExternalVisible := 'False'; ExternalWritable := 'False'} : UDInt;   // Actual time measurement from trigger to get data from camera
         udi_PrevReadingFromCameraTime { ExternalAccessible := 'False'; ExternalVisible := 'False'; ExternalWritable := 'False'} : UDInt;   // Previous time measurement from trigger to get data from camera
         udi_ShortestReadingTime { ExternalAccessible := 'False'; ExternalVisible := 'False'; ExternalWritable := 'False'} : UDInt;   // The shortest time of reading data from camera  (only OK READ)
         udi_LongestReadingTime { ExternalAccessible := 'False'; ExternalVisible := 'False'; ExternalWritable := 'False'} : UDInt;   // The longest time of reading data from camera  (only OK READ)
         udi_AvgReadingTime { ExternalAccessible := 'False'; ExternalVisible := 'False'; ExternalWritable := 'False'} : UDInt;   // Average time of reading data from camera (only OK READ)
         udi_SumOfTimesOkRead { ExternalAccessible := 'False'; ExternalVisible := 'False'; ExternalWritable := 'False'} : UDInt;   // Sum of all OK READ times - for use in average
         udi_ActTimeToNextReady { ExternalAccessible := 'False'; ExternalVisible := 'False'; ExternalWritable := 'False'} : UDInt;   // Time from trigger to get next high state on bit "Trigger Ready" from camera
         si_OK_READ_CounterGeneral { ExternalAccessible := 'False'; ExternalVisible := 'False'; ExternalWritable := 'False'} : UInt;   // Total number of correct readings
         si_TimeOut_CounterGeneral { ExternalAccessible := 'False'; ExternalVisible := 'False'; ExternalWritable := 'False'} : UInt;   // Total number of timeouts
         si_NO_READ_CounterGeneral { ExternalAccessible := 'False'; ExternalVisible := 'False'; ExternalWritable := 'False'} : UInt;   // Total number of NO READ
         si_NO_READ_CounterInRow { ExternalAccessible := 'False'; ExternalVisible := 'False'; ExternalWritable := 'False'} : UInt;   // Number of No READ in a row (after 5 generate error)
      END_STRUCT;
      sw_ErrorCode { ExternalAccessible := 'False'; ExternalVisible := 'False'; ExternalWritable := 'False'} : Word;   // Error code
      sx_BUSY { ExternalAccessible := 'False'; ExternalVisible := 'False'; ExternalWritable := 'False'} : Bool;   // Function is processing data (set with trigger, reset at the end of processing data from the camera)
      sx_OK_READ { ExternalAccessible := 'False'; ExternalVisible := 'False'; ExternalWritable := 'False'} : Bool;   // Correct reading
      sx_NO_READ { ExternalAccessible := 'False'; ExternalVisible := 'False'; ExternalWritable := 'False'} : Bool;   // Camera can't read last barcode
      sx_ErrorTimeOut { ExternalAccessible := 'False'; ExternalVisible := 'False'; ExternalWritable := 'False'} : Bool;   // Begin measuring time with trigger and finish when camera activate "Results Available". Time set up in constants
      "sx_General Fault" { ExternalAccessible := 'False'; ExternalVisible := 'False'; ExternalWritable := 'False'} : Bool;   // Any error set this bit
      sx_ResetResultAvailableBit { ExternalAccessible := 'False'; ExternalVisible := 'False'; ExternalWritable := 'False'} : Bool;   // Bit is used as memory during the reset procedure of "Result available" bit ( it requires communication between the camera and the PLC)
      sx_ResetErrorsInterlocked { ExternalAccessible := 'False'; ExternalVisible := 'False'; ExternalWritable := 'False'} : Bool;   // Bit is used as memory during error reset process.
   END_VAR

   VAR_TEMP
      ti_Trigger_ID : Int;   // ID value of the next trigger to be issued (16-bit integer). Copy of input tag get from camera after decoding UDT bytes (original TriggerID)
      ti_ResultID : Int;   // “Trigger ID” when the trigger that generated these results was. Copy of input tag get from camera after decoding UDT bytes (original ResultID)
      ti_ResultCode : Int;   // Indicates the success or failure of the read that produced these results Copy of input tag get from camera after decoding UDT bytes (original Result Code or "flags")
      ti_ResultLength : Int;   // Actual number of bytes of read data contained in the “Result Data” field (16-bit)  Copy of input tag get from camera after decoding UDT bytes (original Result Code or "flags")
      tx_Decoding : Bool;   // Indicates that the DataMan is decoding an acquired image. The value of the Decoding bit is identical to the value of the Acquiring bit. Both bits are true if an acquisition, or series of acquisitions of the same trigger, is in progress. Copy of input tag get from camera after decoding UDT bytes (original Decoding)
      tx_DecodeComplete : Bool;   // Bit is toggled on the completion of a decode operation when the new results are made available (0 -> 1 or 1 -> 0).  Copy of input tag get from camera after decoding UDT bytes (original Decode complete)
      tx_ResultsBufferOverrun : Bool;   // Indicates that the DataMan has discarded a set of read results because the results Copy of input tag get from camera after decoding UDT bytes (orginal Results Buffer Overrun)
      tx_CameraNoRead : Bool;   // Result Code = 0 -> Camera NO READ code
      tx_CameraOkRead : Bool;   // Result Code = 1 -> Camera READ code
      tx_ResultsAvailable : Bool;   // Indicates that a new set of read results are available, that is, the contents of the Result Data module are valid. Cleared when the results are acknowledged. Copy of input tag get from camera after decoding UDT bytes (orginal Result Available)
   END_VAR

   VAR CONSTANT
      cudi_TimeOut : UDInt := 110;   // Timeout time
      cudi_MaxUDint : UDInt := 4_294_967_295;   // Maximal value of UDint
   END_VAR


BEGIN
	(*

	Version history:
	Date        | Version   | Author             | Remark
	----------------------------------------------------------------------------------------
	08/05/2024   | 0.1       | Grzegorz Czekała    | first release TIA Portal 17 (upd 6)
	11/05/2024   | 0.2       | S. Nieswiec         | removed optional inputs, added barcode string to outputs,
	                                               | changed system commands to equipment control
	25/05/2024   | 0.3       | S. Nieswiec         | Switched IEC timers for FB_TimerOnOffDelay
	27/05/2024   | 0.4       | S. Nieswiec         | Cleaned up code, changed region names
	                                               | TO DO, clean up statistics region, can't just copy paste it higher because statistics brake
	*)


	REGION 1 - Initial

	    REGION 1.1 - Reset Temp variables
	        #ti_Trigger_ID := 0;
	        #ti_ResultID := 0;
	        #ti_ResultCode := 0;
	        #ti_ResultLength := 0;
	        #tx_Decoding := FALSE;
	        #tx_DecodeComplete := FALSE;
	        #tx_ResultsBufferOverrun := FALSE;
	        #tx_CameraOkRead := FALSE;
	        #tx_CameraNoRead := FALSE;
	        #tx_ResultsAvailable := FALSE;
	    END_REGION

	    REGION 1.2 - Timers
	        REGION 1.2.1 - Timeout
	            #sFB_TimerOnOffDelay_TimeOut(iudi_OnDelayTime := #cudi_TimeOut,
	                                         ix_SignalToDelay := #sx_BUSY AND NOT #tx_ResultsAvailable,
	                                         ix_Enable := TRUE);
	        END_REGION

	        REGION 1.2.2 - Results available timeout
	            #sFB_TimerOnOffDelay_ResultsAvailableError(iudi_OnDelayTime := 20,
	                                                       ix_SignalToDelay := #tx_ResultsAvailable,
	                                                       ix_Enable := TRUE);
	        END_REGION
	    END_REGION

	    REGION 1.3 - Triggers
	        #sR_TRIG_Trigger(CLK := #ix_Trigger);  //Rising edge trigger signal
	        //  #sR_TRIG_TriggerReady(CLK := #iUDT_CognexDM260_IN.TriggerReady); lower in code
	        // #sR_TRIG_ResultAvailable(CLK := #"tx_ResultsAvailable");    // lower in code
	        #sR_TRIG_OkReadCounter(CLK := #sx_OK_READ);
	        #sR_TRIG_NoReadCounter(CLK := #sx_NO_READ);
	        #sR_TRIG_ResetStatistics(CLK := #iqUDT_EquipmentControl.Command.ResetData);
	    END_REGION

	    REGION 1.4 - Trigger Enable

	        #qUDT_CognexDM260_OUT.TriggerEnable := TRUE;  // Camera always ready to trigger

	    END_REGION

	END_REGION

	REGION 2. Trigger activation

	    #"tx_ResultsAvailable" := #iUDT_CognexDM260_IN.BYTE_Decoding.%X3; // decoding info from camera "Results Available" (Information on receiving data from the camera regardless of whether the barcode is read or not.)

	    // Activate camera trigger when: camera is ready, input trigger is activated and previous process is completed without errors
	    IF #sR_TRIG_Trigger.Q
	        AND #iUDT_CognexDM260_IN.TriggerReady
	        AND NOT #qUDT_CognexDM260_OUT.Trigger
	        AND NOT #iUDT_CognexDM260_IN.TriggerAck
	        AND NOT #"tx_ResultsAvailable"
	        AND NOT #qUDT_CognexDM260_OUT.ResultsAck
	        AND NOT #sx_BUSY
	        AND NOT #sx_ResetErrorsInterlocked
	    THEN
	        #qUDT_CognexDM260_OUT.Trigger := TRUE;
	        #sx_BUSY := TRUE;   // process in progress
	        #sx_ErrorTimeOut := FALSE;
	        #sx_NO_READ := FALSE;
	        #sx_OK_READ := FALSE;
	        #sw_ErrorCode := 16#0;
	    END_IF;
	END_REGION


	REGION 3 - Handling data received from camera

	    IF #sx_BUSY
	        AND #tx_ResultsAvailable
	        AND NOT #qUDT_CognexDM260_OUT.ResultsAck
	    THEN
	        #qUDT_CognexDM260_OUT.Trigger := FALSE;
	        #qUDT_CognexDM260_OUT.ResultsAck := TRUE;

	        REGION 3.1 - Decoding data

	            // Data decoding is necessary because we receive data from the camera in the form of bytes when we need integers and bit
	            // Decoding byte nr 3
	            #tx_Decoding := #iUDT_CognexDM260_IN.BYTE_Decoding.%X0;
	            #"tx_DecodeComplete" := #iUDT_CognexDM260_IN.BYTE_Decoding.%X1;
	            #"tx_ResultsBufferOverrun" := #iUDT_CognexDM260_IN.BYTE_Decoding.%X2;
	            // #"Results Available" := #iUDT_Cognex260_control."BYTE_Decoding-GeneralFault".%X3;  // This is decoding upper line
	            #"sx_General Fault" := #iUDT_CognexDM260_IN.BYTE_Decoding.%X7;

	            // Trigger ID
	            #ti_Trigger_ID.%B1 := #iUDT_CognexDM260_IN.TriggerID;
	            #ti_Trigger_ID.%B0 := #iUDT_CognexDM260_IN."TriggerID 1";

	            // Result ID
	            #ti_ResultID.%B1 := #iUDT_CognexDM260_IN.ResultID;
	            #ti_ResultID.%B0 := #iUDT_CognexDM260_IN."ResultID 1";

	            // Result Code
	            #ti_ResultCode.%B1 := #iUDT_CognexDM260_IN."Result Code";
	            #ti_ResultCode.%B0 := #iUDT_CognexDM260_IN."Result Code_1";

	            // Result Lenght
	            #ti_ResultLength.%B1 := #iUDT_CognexDM260_IN."Result Length";
	            #ti_ResultLength.%B0 := #iUDT_CognexDM260_IN."Result Length_1";

	            REGION 3.1.1 - Copying last result barcode value

	                // Copy Last Result NO_READ sign
	                #ss_LastResults.DataBarCode[0] := #iUDT_CognexDM260_IN."BarCodeValue[0]-NO_READ_sign";

	                // Copy last result barcode value to DB
	                MOVE_BLK(IN := #iUDT_CognexDM260_IN.BarCodeValue[1],
	                         COUNT := 63,
	                         OUT => #ss_LastResults.DataBarCode[1]);

	                // Marge Bytes to int
	                #ss_LastResults.ID := #ti_ResultID;
	                #ss_LastResults.Flags := #ti_ResultCode;
	                #ss_LastResults.Length := #ti_ResultLength;

	                // For future use conversion from char to string
	                Chars_TO_Strg(Chars := #ss_LastResults.DataBarCode,
	                              pChars := 0,
	                              Cnt := 0,
	                              Strg => #ss_LastResults.DataBarCodeString);
	                #qs_Barcode := #ss_LastResults.DataBarCodeString;
	            END_REGION

	        END_REGION

	        REGION 3.2  No READ // When NO_READ this bit is activate (is set until new trigger)

	            // Check when get new data if there is "!"
	            IF #qUDT_CognexDM260_OUT.ResultsAck AND #ss_LastResults.DataBarCode[0] = '!'
	            THEN
	                #sx_NO_READ := TRUE;
	                #sx_OK_READ := FALSE;
	            END_IF;

	            IF #qUDT_CognexDM260_OUT.ResultsAck AND #ss_LastResults.DataBarCode[0] <> '!'
	            THEN
	                #sx_NO_READ := FALSE;
	                #sx_OK_READ := TRUE;
	            END_IF;

	            //Addidtional data from camera
	            #tx_CameraOkRead := #ti_ResultCode.%X0 AND #qUDT_CognexDM260_OUT.ResultsAck;
	            #tx_CameraNoRead := NOT #ti_ResultCode.%X0 AND #qUDT_CognexDM260_OUT.ResultsAck;

	        END_REGION
	    END_IF;

	    REGION 3.3  End of reading procedure
	        //Resets bits  is READY TO next trigger
	        IF #sx_BUSY
	            AND #qUDT_CognexDM260_OUT.ResultsAck
	            AND NOT #"tx_ResultsAvailable"
	        THEN
	            #qUDT_CognexDM260_OUT.ResultsAck := FALSE;
	            #sx_BUSY := FALSE;
	        END_IF;

	    END_REGION
	END_REGION


	REGION 4 - Statistics


	    REGION 4.1  Time statistics

	        ////////////////////////////////// Time measured from trigger to receiving a response "Results Available".

	        #sR_TRIG_ResultAvailable(CLK := #"tx_ResultsAvailable");
	        #sR_TRIG_StatisticActCycleTime(CLK := #sR_TRIG_ResultAvailable.Q OR #sx_ErrorTimeOut);


	        IF #sR_TRIG_StatisticActCycleTime.Q  // Sending the time only once in the event of receiving data or exceeding the timeout.
	        THEN
	            #ss_Statistic.udi_PrevReadingFromCameraTime := #ss_Statistic.udi_ActReadingFromCameraTime;
	            #ss_Statistic.udi_ActReadingFromCameraTime := LREAL_TO_UDINT(#sFB_TimerOnOffDelay_ActTimeToNextReady.qlr_ActualTime);
	            #sFB_TimerOnOffDelay_ActReadingFromCameraTime.ix_SignalToDelay := FALSE;
	        END_IF;

	        REGION 4.1.1 Longest, shortest and average reading time

	            // Statistics include only OK_READ process
	            IF #sR_TRIG_ResultAvailable.Q AND #sx_OK_READ
	            THEN

	                // Chceck the longest time
	                IF #ss_Statistic.udi_ActReadingFromCameraTime > #ss_Statistic.udi_LongestReadingTime
	                THEN
	                    #ss_Statistic.udi_LongestReadingTime := #ss_Statistic.udi_ActReadingFromCameraTime;

	                END_IF;

	                // When PLC startup the shortest time is 0ms, so we put there other start shortest time value
	                IF #ss_Statistic.udi_ShortestReadingTime < 1
	                THEN
	                    #ss_Statistic.udi_ShortestReadingTime := #ss_Statistic.udi_ActReadingFromCameraTime;
	                END_IF;

	                // Chceck the shortest time
	                IF (#ss_Statistic.udi_ActReadingFromCameraTime < #ss_Statistic.udi_ShortestReadingTime)
	                THEN

	                    #ss_Statistic.udi_ShortestReadingTime := #ss_Statistic.udi_ActReadingFromCameraTime;
	                END_IF;

	                // Calculate average time of OK_READs
	                #ss_Statistic.udi_SumOfTimesOkRead := #ss_Statistic.udi_SumOfTimesOkRead + #ss_Statistic.udi_ActReadingFromCameraTime;
	                #ss_Statistic.udi_AvgReadingTime := #ss_Statistic.udi_SumOfTimesOkRead / #ss_Statistic.si_OK_READ_CounterGeneral;

	            END_IF;
	        END_REGION

	        REGION 4.1.2 Time from trigger to ResultsAvailable

	            IF #sx_BUSY AND NOT #tx_ResultsAvailable THEN
	                #sFB_TimerOnOffDelay_ActReadingFromCameraTime.ix_SignalToDelay := TRUE;
	            END_IF;

	            #sFB_TimerOnOffDelay_ActReadingFromCameraTime(iudi_OnDelayTime := #cudi_MaxUDint,
	                                                          ix_Enable := TRUE);

	            //Time measured from trigger to receiving a response "Trigger ready".
	            #sR_TRIG_TriggerReady(CLK := #iUDT_CognexDM260_IN.TriggerReady);

	            IF #sx_BUSY THEN
	                #sFB_TimerOnOffDelay_ActTimeToNextReady.ix_SignalToDelay := TRUE;
	            END_IF;

	            IF #sR_TRIG_TriggerReady.Q OR #sx_ErrorTimeOut
	            THEN
	                #ss_Statistic.udi_ActTimeToNextReady := LREAL_TO_UDINT(#sFB_TimerOnOffDelay_ActTimeToNextReady.qlr_ActualTime);
	                #sFB_TimerOnOffDelay_ActTimeToNextReady.ix_SignalToDelay := FALSE;
	            END_IF;

	            #sFB_TimerOnOffDelay_ActTimeToNextReady(iudi_OnDelayTime := #cudi_MaxUDint,
	                                                    ix_Enable := TRUE);
	        END_REGION
	    END_REGION


	    REGION 4.2 - Count statistics
	        REGION 4.2.1 - OK_READ

	            IF #sR_TRIG_OkReadCounter.Q
	            THEN
	                #ss_Statistic.si_OK_READ_CounterGeneral += 1;
	            END_IF;
	        END_REGION

	        REGION 4.2.2 -  NO_READ and NO_READ in row

	            IF #sx_OK_READ
	            THEN
	                #ss_Statistic.si_NO_READ_CounterInRow := 0;
	            END_IF;

	            IF #sR_TRIG_NoReadCounter.Q
	            THEN
	                #ss_Statistic.si_NO_READ_CounterGeneral += 1;
	                #ss_Statistic.si_NO_READ_CounterInRow += 1;
	            END_IF;
	        END_REGION
	    END_REGION

	    REGION 4.3 - Reset statistics

	        // Reset all statistic
	        IF #sR_TRIG_ResetStatistics.Q
	        THEN
	            #ss_Statistic.udi_ActReadingFromCameraTime := 0;
	            #ss_Statistic.udi_PrevReadingFromCameraTime := 0;
	            #ss_Statistic.udi_ShortestReadingTime := 0;
	            #ss_Statistic.udi_SumOfTimesOkRead := 0;
	            #ss_Statistic.udi_LongestReadingTime := 0;
	            #ss_Statistic.udi_ActTimeToNextReady := 0;
	            #ss_Statistic.udi_AvgReadingTime := 0;
	            #ss_Statistic.si_OK_READ_CounterGeneral := 0;
	            #ss_Statistic.si_TimeOut_CounterGeneral := 0;
	            #ss_Statistic.si_NO_READ_CounterInRow := 0;
	            #ss_Statistic.si_NO_READ_CounterGeneral := 0;
	        END_IF;
	    END_REGION

	END_REGION

	REGION 5 - End of reading procedure

	    IF #sx_BUSY
	        AND #qUDT_CognexDM260_OUT.ResultsAck
	        AND NOT #"tx_ResultsAvailable"
	    THEN
	        #qUDT_CognexDM260_OUT.ResultsAck := FALSE;
	        #sx_BUSY := FALSE;

	    END_IF;

	END_REGION

	REGION 6 - Errors

	    REGION 4.1 - Timeout

	        IF #sFB_TimerOnOffDelay_TimeOut.qx_DelayedSignal THEN
	            #sx_ErrorTimeOut := TRUE;
	        END_IF;

	        IF #sR_TRIG_TimeOutCounter.Q
	        THEN
	            #ss_Statistic.si_TimeOut_CounterGeneral += 1;
	        END_IF;
	    END_REGION

	    REGION 4.2 - Results available blocked

	        IF #sFB_TimerOnOffDelay_ResultsAvailableError.qx_DelayedSignal
	        THEN
	            #"sx_General Fault" := TRUE;
	            #sw_ErrorCode := 16#800B;             // Bit from camera "Result available" blocked
	            #sx_ResetErrorsInterlocked := TRUE;  // Start procedure of reset bit Results Available
	        END_IF;

	        IF #sx_ErrorTimeOut AND #"tx_ResultsAvailable"
	        THEN
	            #sx_ResetErrorsInterlocked := TRUE;  // Reset bit Results Available
	        END_IF;
	    END_REGION

	    REGION 4.3 - Error codes

	        REGION 4.3.1 - Timeout
	            IF #sx_ErrorTimeOut
	            THEN
	                #"sx_General Fault" := TRUE;
	                #sw_ErrorCode := 16#800A;
	            END_IF;
	        END_REGION

	        REGION 4.3.2 - No read
	            IF #sx_NO_READ
	            THEN
	                #"sx_General Fault" := TRUE;
	                #sw_ErrorCode := 16#800C;     // NO READ
	            END_IF;
	        END_REGION

	        REGION 4.3.3 - Five no read in row
	            IF #ss_Statistic.si_NO_READ_CounterInRow >= 5
	            THEN
	                #"sx_General Fault" := TRUE;
	                #sw_ErrorCode := 16#805C;    // 5 NO READ in row
	            END_IF;
	        END_REGION

	        REGION 4.3.4 - Empty data from camera
	            IF #qUDT_CognexDM260_OUT.ResultsAck AND #ss_LastResults.DataBarCode[0] = '$00'
	            THEN
	                #"sx_General Fault" := TRUE;
	                #sw_ErrorCode := 16#80C0;    // Empty data from camera
	            END_IF;
	        END_REGION

	        REGION 4.3.5 - Writing error code to ouput

	            #qw_RetVal := #sw_ErrorCode;

	        END_REGION
	    END_REGION
	END_REGION

	REGION 7 - Errors reset

	    REGION 6.1 - General
	        IF #iqUDT_EquipmentControl.Command.Reset THEN
	            #ss_Statistic.si_TimeOut_CounterGeneral := 0;
	            #ss_Statistic.si_NO_READ_CounterInRow := 0;

	            #sx_BUSY := FALSE;
	            #qUDT_CognexDM260_OUT.ResultsAck := FALSE;
	            #"sx_General Fault" := TRUE;
	            #sw_ErrorCode := 16#0000;

	            #sx_ResetErrorsInterlocked := TRUE;
	        END_IF;
	    END_REGION

	    REGION 6.2 Reset "Result Available" and Trigger Ack bit from camera

	        // To clear the bit "#Results Available" from camera, it is necessary to SET the bit "ResultsAck" and wait for confirmation from the camera.
	        IF #sx_ResetResultAvailableBit AND NOT #"tx_ResultsAvailable"
	        THEN
	            #sx_ResetResultAvailableBit := FALSE;
	            #qUDT_CognexDM260_OUT.ResultsAck := FALSE;
	            #qUDT_CognexDM260_OUT.Trigger := FALSE;
	        END_IF;

	        IF #sx_ResetErrorsInterlocked AND #"tx_ResultsAvailable"
	        THEN
	            #qUDT_CognexDM260_OUT.ResultsAck := TRUE;
	            #sx_ResetResultAvailableBit := TRUE;
	        END_IF;


	        IF #sx_ResetErrorsInterlocked AND NOT #"tx_ResultsAvailable"
	        THEN
	            #sx_ResetErrorsInterlocked := FALSE;
	        END_IF;

	    END_REGION
	END_REGION



END_FUNCTION_BLOCK

